Staubli VAL3: ASCIItoNum.pgx

public program ASCIItoNum(num& x_nAsc (dimensions=1), num& x_nNum (dimensions=1))
begin

  //将ASCII码（十进制）转换成十进制数字（用于求出十六进制数每位上的数字）
  if x_nAsc>=48 and x_nAsc<=57
    x_nNum=x_nAsc-48
  elseIf x_nAsc>=65 and x_nAsc<=70
    x_nNum=x_nAsc-65+10
  endIf

end
